FUNCTION F_SineFunction_primary : LREAL
VAR_INPUT
	fTime 				: LREAL;
END_VAR
VAR_OUTPUT
	fSineSignal 		: LREAL;
END_VAR
VAR
	u					: LREAL;
	ft_ENV				: LREAL;
	y					: LREAL;
	
END_VAR

ft_ENV := G_Engineer_HMI.ft_ENV;

u := fTime/ft_ENV;

IF u > 1.0 THEN
	u := 1.0;
END_IF

y := (3.0*u*u) - (2.0*u*u*u);

fSineSignal := y* G_Engineer_HMI.fAmp * SIN(2.0 * PI * G_Engineer_HMI.fFreq * fTime) + G_Engineer_HMI.fSinemidpoint;

END_FUNCTION

(* stored: Version 1.1.0.1
   POU F_SineFunction_primary: Id {36c62ab0-3dfd-4d51-af4c-aadf4d024ecd}, SpecialFunc None *)
